(* CoDeSys 2.3.9.52 project: dom1a.pro *)
(* Libraries: Standard.lib 8.11.10 11:37:48, SYSLIBCALLBACK.LIB 8.11.10 11:37:48 *)

(* PLC configuration (modules and I/O channels)
0750-0430 8 DI 24 V DC 3.0ms [Type_1_8_Channels] node 0, in %IB0 out %QB0 {INTTypePAAssignment = PLC; INTTypeModule = plugged}
  AT %IX0.0 [BOOLOnX_I] Ch_1 Digital input
  AT %IX0.1 [BOOLOnX_I] Ch_2 Digital input
  AT %IX0.2 [BOOLOnX_I] Ch_3 Digital input
  AT %IX0.3 [BOOLOnX_I] Ch_4 Digital input
  AT %IX0.4 [BOOLOnX_I] Ch_5 Digital input
  AT %IX0.5 [BOOLOnX_I] Ch_6 Digital input
  AT %IX0.6 [BOOLOnX_I] Ch_7 Digital input
  AT %IX0.7 [BOOLOnX_I] Ch_8 Digital input
0750-0430 8 DI 24 V DC 3.0ms [Type_1_8_Channels] node 0, in %IB0 out %QB0 {INTTypePAAssignment = PLC; INTTypeModule = plugged}
  AT %IX0.8 [BOOLOnX_I] Ch_1 Digital input
  AT %IX0.9 [BOOLOnX_I] Ch_2 Digital input
  AT %IX0.10 [BOOLOnX_I] Ch_3 Digital input
  AT %IX0.11 [BOOLOnX_I] Ch_4 Digital input
  AT %IX0.12 [BOOLOnX_I] Ch_5 Digital input
  AT %IX0.13 [BOOLOnX_I] Ch_6 Digital input
  AT %IX0.14 [BOOLOnX_I] Ch_7 Digital input
  AT %IX0.15 [BOOLOnX_I] Ch_8 Digital input
0750-0430 8 DI 24 V DC 3.0ms [Type_1_8_Channels] node 0, in %IB1 out %QB0 {INTTypePAAssignment = PLC; INTTypeModule = plugged}
  AT %IX1.0 [BOOLOnX_I] Ch_1 Digital input
  AT %IX1.1 [BOOLOnX_I] Ch_2 Digital input
  AT %IX1.2 [BOOLOnX_I] Ch_3 Digital input
  AT %IX1.3 [BOOLOnX_I] Ch_4 Digital input
  AT %IX1.4 [BOOLOnX_I] Ch_5 Digital input
  AT %IX1.5 [BOOLOnX_I] Ch_6 Digital input
  AT %IX1.6 [BOOLOnX_I] Ch_7 Digital input
  AT %IX1.7 [BOOLOnX_I] Ch_8 Digital input
0750-0430 8 DI 24 V DC 3.0ms [Type_1_8_Channels] node 0, in %IB2 out %QB0 {INTTypePAAssignment = PLC; INTTypeModule = plugged}
  AT %IX1.8 [BOOLOnX_I] Ch_1 Digital input
  AT %IX1.9 [BOOLOnX_I] Ch_2 Digital input
  AT %IX1.10 [BOOLOnX_I] Ch_3 Digital input
  AT %IX1.11 [BOOLOnX_I] Ch_4 Digital input
  AT %IX1.12 [BOOLOnX_I] Ch_5 Digital input
  AT %IX1.13 [BOOLOnX_I] Ch_6 Digital input
  AT %IX1.14 [BOOLOnX_I] Ch_7 Digital input
  AT %IX1.15 [BOOLOnX_I] Ch_8 Digital input
0750-0430 8 DI 24 V DC 3.0ms [Type_1_8_Channels] node 0, in %IB3 out %QB0 {INTTypePAAssignment = PLC; INTTypeModule = plugged}
  AT %IX2.0 [BOOLOnX_I] Ch_1 Digital input
  AT %IX2.1 [BOOLOnX_I] Ch_2 Digital input
  AT %IX2.2 [BOOLOnX_I] Ch_3 Digital input
  AT %IX2.3 [BOOLOnX_I] Ch_4 Digital input
  AT %IX2.4 [BOOLOnX_I] Ch_5 Digital input
  AT %IX2.5 [BOOLOnX_I] Ch_6 Digital input
  AT %IX2.6 [BOOLOnX_I] Ch_7 Digital input
  AT %IX2.7 [BOOLOnX_I] Ch_8 Digital input
0750-0430 8 DI 24 V DC 3.0ms [Type_1_8_Channels] node 0, in %IB4 out %QB0 {INTTypePAAssignment = PLC; INTTypeModule = plugged}
  AT %IX2.8 [BOOLOnX_I] Ch_1 Digital input
  AT %IX2.9 [BOOLOnX_I] Ch_2 Digital input
  AT %IX2.10 [BOOLOnX_I] Ch_3 Digital input
  AT %IX2.11 [BOOLOnX_I] Ch_4 Digital input
  AT %IX2.12 [BOOLOnX_I] Ch_5 Digital input
  AT %IX2.13 [BOOLOnX_I] Ch_6 Digital input
  AT %IX2.14 [BOOLOnX_I] Ch_7 Digital input
  AT %IX2.15 [BOOLOnX_I] Ch_8 Digital input
0750-0430 8 DI 24 V DC 3.0ms [Type_1_8_Channels] node 0, in %IB5 out %QB0 {INTTypePAAssignment = PLC; INTTypeModule = plugged}
  AT %IX3.0 [BOOLOnX_I] Ch_1 Digital input
  AT %IX3.1 [BOOLOnX_I] Ch_2 Digital input
  AT %IX3.2 [BOOLOnX_I] Ch_3 Digital input
  AT %IX3.3 [BOOLOnX_I] Ch_4 Digital input
  AT %IX3.4 [BOOLOnX_I] Ch_5 Digital input
  AT %IX3.5 [BOOLOnX_I] Ch_6 Digital input
  AT %IX3.6 [BOOLOnX_I] Ch_7 Digital input
  AT %IX3.7 [BOOLOnX_I] Ch_8 Digital input
0750-0530 8 DO 24 V DC 0.5A [Type_10_8_Channels] node 0, in %IB6 out %QB0 {INTTypePAAssignment = PLC; INTTypeModule = plugged}
  AT %QX0.0 [BOOLOnX_Q] Ch_1 Digital output
  AT %QX0.1 [BOOLOnX_Q] Ch_2 Digital output
  AT %QX0.2 [BOOLOnX_Q] Ch_3 Digital output
  AT %QX0.3 [BOOLOnX_Q] Ch_4 Digital output
  AT %QX0.4 [BOOLOnX_Q] Ch_5 Digital output
  AT %QX0.5 [BOOLOnX_Q] Ch_6 Digital output
  AT %QX0.6 [BOOLOnX_Q] Ch_7 Digital output
  AT %QX0.7 [BOOLOnX_Q] Ch_8 Digital output
0750-0530 8 DO 24 V DC 0.5A [Type_10_8_Channels] node 0, in %IB7 out %QB0 {INTTypePAAssignment = PLC; INTTypeModule = plugged}
  AT %QX0.8 [BOOLOnX_Q] Ch_1 Digital output
  AT %QX0.9 [BOOLOnX_Q] Ch_2 Digital output
  AT %QX0.10 [BOOLOnX_Q] Ch_3 Digital output
  AT %QX0.11 [BOOLOnX_Q] Ch_4 Digital output
  AT %QX0.12 [BOOLOnX_Q] Ch_5 Digital output
  AT %QX0.13 [BOOLOnX_Q] Ch_6 Digital output
  AT %QX0.14 [BOOLOnX_Q] Ch_7 Digital output
  AT %QX0.15 [BOOLOnX_Q] Ch_8 Digital output
0750-0530 8 DO 24 V DC 0.5A [Type_10_8_Channels] node 0, in %IB7 out %QB1 {INTTypePAAssignment = PLC; INTTypeModule = plugged}
  AT %QX1.0 [BOOLOnX_Q] Ch_1 Digital output
  AT %QX1.1 [BOOLOnX_Q] Ch_2 Digital output
  AT %QX1.2 [BOOLOnX_Q] Ch_3 Digital output
  AT %QX1.3 [BOOLOnX_Q] Ch_4 Digital output
  AT %QX1.4 [BOOLOnX_Q] Ch_5 Digital output
  AT %QX1.5 [BOOLOnX_Q] Ch_6 Digital output
  AT %QX1.6 [BOOLOnX_Q] Ch_7 Digital output
  AT %QX1.7 [BOOLOnX_Q] Ch_8 Digital output
0750-0530 8 DO 24 V DC 0.5A [Type_10_8_Channels] node 0, in %IB7 out %QB2 {INTTypePAAssignment = PLC; INTTypeModule = plugged}
  AT %QX1.8 [BOOLOnX_Q] Ch_1 Digital output
  AT %QX1.9 [BOOLOnX_Q] Ch_2 Digital output
  AT %QX1.10 [BOOLOnX_Q] Ch_3 Digital output
  AT %QX1.11 [BOOLOnX_Q] Ch_4 Digital output
  AT %QX1.12 [BOOLOnX_Q] Ch_5 Digital output
  AT %QX1.13 [BOOLOnX_Q] Ch_6 Digital output
  AT %QX1.14 [BOOLOnX_Q] Ch_7 Digital output
  AT %QX1.15 [BOOLOnX_Q] Ch_8 Digital output
0750-0530 8 DO 24 V DC 0.5A [Type_10_8_Channels] node 0, in %IB7 out %QB3 {INTTypePAAssignment = PLC; INTTypeModule = plugged}
  AT %QX2.0 [BOOLOnX_Q] Ch_1 Digital output
  AT %QX2.1 [BOOLOnX_Q] Ch_2 Digital output
  AT %QX2.2 [BOOLOnX_Q] Ch_3 Digital output
  AT %QX2.3 [BOOLOnX_Q] Ch_4 Digital output
  AT %QX2.4 [BOOLOnX_Q] Ch_5 Digital output
  AT %QX2.5 [BOOLOnX_Q] Ch_6 Digital output
  AT %QX2.6 [BOOLOnX_Q] Ch_7 Digital output
  AT %QX2.7 [BOOLOnX_Q] Ch_8 Digital output
  AT %QX2.8 [BOOLOnX_Q] Ch_1 Digital output
  AT %QX2.9 [BOOLOnX_Q] Ch_2 Digital output
  AT %QX2.10 [BOOLOnX_Q] Ch_3 Digital output
  AT %QX2.11 [BOOLOnX_Q] Ch_4 Digital output
  AT %QX2.12 [BOOLOnX_Q] Ch_5 Digital output
  AT %QX2.13 [BOOLOnX_Q] Ch_6 Digital output
  AT %QX2.14 [BOOLOnX_Q] Ch_7 Digital output
  AT %QX2.15 [BOOLOnX_Q] Ch_8 Digital output
Fieldbus variables [FB_VARS] node 1, in %IB0 out %QB0
Flag variables [FLAG_VARS] node 2, in %IB0 out %QB0
Modbus-Master [MB_MASTER] node 3, in %IB0 out %QB0
*)

(* Task configuration *)
TASK clock1s (PRIORITY := 1, INTERVAL := T#1000ms);
	clock1s();
END_TASK
TASK loop (PRIORITY := 2);
	PLC_PRG();
END_TASK

(* POU clock1s, ST *)
PROGRAM clock1s
VAR
	test0 AT %QX0.0:BOOL;
	test1 AT %QX0.1:BOOL;
	test2 AT %QX0.2:BOOL;
	test3 AT %QX0.3:BOOL;
	test4 AT %QX0.4:BOOL;
	test5 AT %QX0.5:BOOL;
	test6 AT %QX0.6:BOOL;
	test7 AT %QX0.7:BOOL;
	tmp:BOOL;
END_VAR
tmp := test0;
test0:=test7;
test7:=test6;
test6:=test5;
test5:=test4;
test4:=test3;
test3:=test2;
test2:=test1;
test1:=tmp;
END_PROGRAM

(* POU PLC_PRG, ST *)
PROGRAM PLC_PRG
VAR
	test0 AT %QX0.0:BOOL;
	test1 AT %QX0.1:BOOL;
	test2 AT %QX0.2:BOOL;
	test3 AT %QX0.3:BOOL;
	test4 AT %QX0.4:BOOL;
	test5 AT %QX0.5:BOOL;
	test6 AT %QX0.6:BOOL;
	test7 AT %QX0.7:BOOL;
	firstLoop:BOOL;

	ww: BOOL;
END_VAR
IF NOT firstLoop THEN
	firstLoop:=1;
	start();
END_IF

;
END_PROGRAM

(* POU start, ST *)
PROGRAM start
VAR

	test0 AT %QX0.0:BOOL;
END_VAR
test0 := 1;
END_PROGRAM

(* POU Interrupt_0, ST *)
PROGRAM Interrupt_0
VAR
END_VAR
 %QX0.0 := 1;
END_PROGRAM

(* POU Configuration/MODBUS_CONFIGURATION, ST *)
PROGRAM MODBUS_CONFIGURATION        
VAR                                
END_VAR                            
(*                                 
   <?xml version="1.0" encoding="UTF-16" standalone="yes"?>
<network xml_structure_version="1" xml_feature_version="1">
	<generator_settings minRTUTaskCycleTimeMs="5" minEthaskCycleTimeMs="5" ethSlaveMultiplier="0.1" rtuInterfaceMultiplier="0.1" taskGeneration="true"/>
</network>
                              
*)                                 
;                                  
END_PROGRAM
